{attribute addProperty BoxType "EL7221-0000-0021"}
{attribute addProperty Id "FB_PositionAT %I*FB_Position_BA8AA9F03240DRV_StatuswordAT %I*DRV_Statusword_53CBCECC1620DRV_ControlwordAT %Q*DRV_Controlword_417617681620DRV_Target_velocityAT %Q*DRV_Target_velocity_53A88AB03240WcStateAT %I*WcState_F855686C1620InfoDataAT %I*InfoData_AEB17F4D152190"}
{attribute addProperty CRC "2144119762"}
{attribute addProperty SizeInBites "264"}
{attribute addProperty SizeInBytes "33"}
TYPE EL7221_5C474831 :
STRUCT
	{attribute addProperty Name "FB_Position"}
	FB_Position : FB_Position_BA8AA9F0;
	{attribute addProperty Name "DRV_Statusword"}
	DRV_Statusword : DRV_Statusword_53CBCECC;
	{attribute addProperty Name "DRV_Controlword"}
	DRV_Controlword : DRV_Controlword_41761768;
	{attribute addProperty Name "DRV_Target_velocity"}
	DRV_Target_velocity : DRV_Target_velocity_53A88AB0;
	{attribute addProperty Name "WcState"}
	WcState : WcState_F855686C;
	{attribute addProperty Name "InfoData"}
	InfoData : InfoData_AEB17F4D;
END_STRUCT
END_TYPE

(* stored: Version 1.2.0.0, ProductVersion 3.1.4024.9
   DUT EL7221_5C474831: Id {2d71b248-8299-48a6-b859-9eac4c10090f} *)
